# B&R Automation Studio project Ironer_Line
Automation Studio 4.7.2.98; technology packages: mapp 5.11.2, mappView 5.11.3

## Configuration Config1

CPU X20CP0484, AutomationRuntime B4.73, Build 4.1.2, Safety 0.0, Vc V4.44.0

### Task classes (Cpu.sw)
```
Cyclic#4 (cycle 100000 us, tolerance 100000 us):
  Failsafe <- Failsafe.prg
Cyclic#7 (cycle 1000000 us, tolerance 1000000 us):
  Data_log_p <- Data_log_prog.prg
Binaries: arsvcreg, TCData, udbdef, mvLoader, ashwd, sysconf, ashwac, asfw, arconfig, Role, Config, iomap, User, ArCoal, ArFlatPrv, OpcUaMap
Libraries: AsZip, FileIO, runtime, MpData, DataObj, sys_lib, brsystem, MpBase, astime, AsIODiag, asieccon, arssl
```

### Hardware
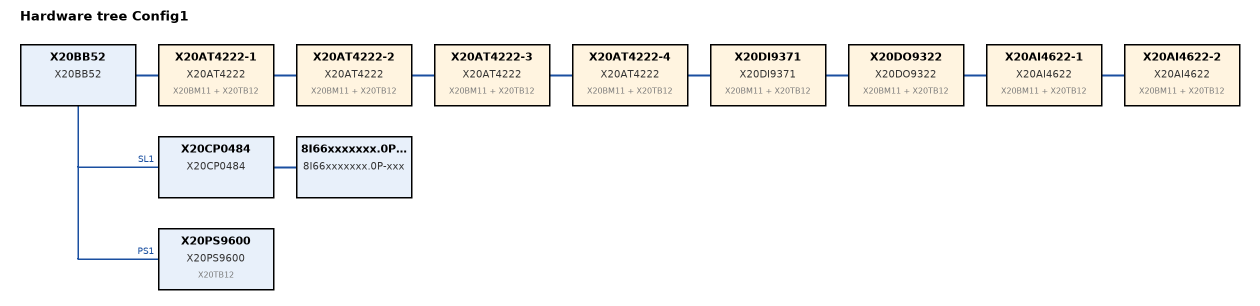
```
8I66xxxxxxx.0P-xxx : 8I66xxxxxxx.0P-xxx v2.3.0.0  [PLK1 -> X20CP0484.IF3 [Cable Type=PowerlinkCable, Length=10, Version=1.0.0.2]]
  FunctionModel = Standard
  Supervision = off
  UnitOfSetpoint = Rpm
  IOM_AIDP1 = ULN
  IOM_AIDP2 = RFR_D
  IOM_AIDP3 = UOP
  IOM_AIDP4 = LCR
  Sel_NameplateMask = MANU
  Cfg_NSP = 2853
  Cfg_UNS = 400
  Cfg_NCR = 25
  Cfg_COS = 80
  Cfg_NPR = 110
X20AI4622-1 : X20AI4622 v1.0.5.0  [SS1 -> X20TB12g.SS; SL -> X20BM11f.SL1]
  Supervision = off
  ChannelType01 = 4 to 20mA
X20AI4622-2 : X20AI4622 v1.0.5.0  [SS1 -> X20TB12h.SS; SL -> X20BM11g.SL1]
  Supervision = off
  ChannelType01 = 4 to 20mA
  ChannelType02 = 4 to 20mA
  ChannelType03 = 4 to 20mA
X20AT4222-1 : X20AT4222 v1.2.2.0  [SS1 -> X20TB12a.SS; SL -> X20BM11.SL1]
  FunctionModel = FunctionModel001
  Supervision = off
  SensorType02 = off
  SensorType03 = off
X20AT4222-2 : X20AT4222 v1.2.2.0  [SS1 -> X20TB12b.SS; SL -> X20BM11a.SL1]
  FunctionModel = FunctionModel001
  Supervision = off
  SensorType03 = off
  SensorType04 = off
X20AT4222-3 : X20AT4222 v1.2.2.0  [SS1 -> X20TB12c.SS; SL -> X20BM11b.SL1]
  FunctionModel = FunctionModel001
  Supervision = off
  SensorType03 = off
  SensorType04 = off
X20AT4222-4 : X20AT4222 v1.2.2.0  [SS1 -> X20TB12d.SS; SL -> X20BM11c.SL1]
  FunctionModel = FunctionModel001
  Supervision = off
  SensorType03 = off
  SensorType04 = off
X20BB52 : X20BB52 v1.1.0.0
X20BM11 : X20BM11 v1.0.0.1  [X2X1 -> X20BB52.IF6]
X20BM11a : X20BM11 v1.0.0.1  [X2X1 -> X20BM11.X2X2]
X20BM11b : X20BM11 v1.0.0.1  [X2X1 -> X20BM11a.X2X2]
X20BM11c : X20BM11 v1.0.0.1  [X2X1 -> X20BM11b.X2X2]
X20BM11d : X20BM11 v1.0.0.1  [X2X1 -> X20BM11c.X2X2]
X20BM11e : X20BM11 v1.0.0.1  [X2X1 -> X20BM11d.X2X2]
X20BM11f : X20BM11 v1.0.0.1  [X2X1 -> X20BM11e.X2X2]
X20BM11g : X20BM11 v1.0.0.1  [X2X1 -> X20BM11f.X2X2]
X20CP0484 : X20CP0484 v1.2.0.0  [SL -> X20BB52.SL1]
  Connector IF2:
    ActivateDevice = 1
    Mode = Manual
    InternetAddress = 10.0.0.2
    SubnetMask = 255.255.255.0
    InaNodeNumber = 0
  ConfigurationID = EIT5Projekt1_Config1
  UserPartitionSize = 100
  Simulation = 1
  TimerDeviceType = SWIOTIMER
  Cyclic1Duration = 10000
  Cyclic1Tolerance = 10000
  Cyclic2Duration = 20000
  Cyclic2Tolerance = 20000
  Cyclic3Duration = 50000
  Cyclic3Tolerance = 50000
  Cyclic4Duration = 100000
  Cyclic4Tolerance = 100000
  Cyclic5Duration = 200000
  Cyclic5Tolerance = 200000
  Cyclic6Duration = 500000
  Cyclic6Tolerance = 500000
  Cyclic7Duration = 1000000
  Cyclic7Tolerance = 1000000
  Cyclic8Duration = 10000
  Cyclic8Tolerance = 30000000
  FileDevice1
  FileDeviceName1 = PLC_user
  FileDevicePath1 = F:\
  FileDevice2
  FileDeviceName2 = PC_temp
  FileDevicePath2 = C:\temp\
  FtpUser1
  FtpUsername1 = admin
  FtpUserPassword1 = cwHDI+xQYJGOTM1OUrZCZFPwGlAu3H/MLCABeDPRdiI=  // password=admin
  FtpUserSalt1 = YD4DOUwF
  FTPAccessRight1 = 0
  FTPdevice1 = ALL
  ActivateOpcUa = 1
  OpcUaInformationModels_PV_Version = 1
X20DI9371 : X20DI9371 v1.0.2.0  [SS1 -> X20TB12e.SS; SL -> X20BM11d.SL1]
  Supervision = off
X20DO9322 : X20DO9322 v1.0.3.0  [SS1 -> X20TB12f.SS; SL -> X20BM11e.SL1]
  Supervision = off
X20PS9600 : X20PS9600 v1.0.1.0  [PS -> X20BB52.PS1; SS1 -> X20TB12.SS]
  Supervision = off
X20TB12 : X20TB12 v1.0.0.0
X20TB12a : X20TB12 v1.0.0.0
X20TB12b : X20TB12 v1.0.0.0
X20TB12c : X20TB12 v1.0.0.0
X20TB12d : X20TB12 v1.0.0.0
X20TB12e : X20TB12 v1.0.0.0
X20TB12f : X20TB12 v1.0.0.0
X20TB12g : X20TB12 v1.0.0.0
X20TB12h : X20TB12 v1.0.0.0
```

### IoMap.iom - X20CP0484/IoMap.iom
```iecst
VAR_CONFIG
	::T_tank AT %IW."X20AT4222-1".Temperature01;
	::inverter.CTRL_set AT %QW."8I66xxxxxxx.0P-xxx".CMDD_Output;
	::inverter.RPM_set AT %QW."8I66xxxxxxx.0P-xxx".LFRD_Output;
	::inverter.RPM_actual AT %IW."8I66xxxxxxx.0P-xxx".RFRD_Input;
	::inverter.freq AT %IW."8I66xxxxxxx.0P-xxx".RFR_Input;
	::inverter.voltage AT %IW."8I66xxxxxxx.0P-xxx".UOP_Input;
	::inverter.current AT %IW."8I66xxxxxxx.0P-xxx".LCR_Input;
	::inverter.DC AT %IW."8I66xxxxxxx.0P-xxx".ULN_Input;
	::inverter.error_code AT %IW."8I66xxxxxxx.0P-xxx".ERRD_Input;
	::inverter.CTRL_actual AT %IW."8I66xxxxxxx.0P-xxx".ETAD_Input;
	::inverter.RPM_after_ramp AT %IW."8I66xxxxxxx.0P-xxx".FROD_Input;
	::mulde_3.T_out AT %IW."X20AT4222-4".Temperature02;
	::mulde_3.T_in AT %IW."X20AT4222-4".Temperature01;
	::mulde_1.T_in AT %IW."X20AT4222-2".Temperature01;
	::mulde_2.T_out AT %IW."X20AT4222-3".Temperature02;
	::mulde_2.T_in AT %IW."X20AT4222-3".Temperature01;
	::mulde_1.T_out AT %IW."X20AT4222-2".Temperature02;
	::heater AT %QX."X20DO9322".DigitalOutput01;
	::T_ambient AT %IW."X20AT4222-1".Temperature04;
	::flow_cooling_water AT %IW."X20AI4622-1".AnalogInput01;
	::p_pumpe.before AT %IW."X20AI4622-2".AnalogInput01;
	::p_pumpe.after AT %IW."X20AI4622-2".AnalogInput02;
	::p_last AT %IW."X20AI4622-2".AnalogInput03;
END_VAR
```

### Config.mpdatarecorder - X20CP0484/mappServices/Config.mpdatarecorder
```
Element gDataRecorder (Type=mpdatarecorder)
  DataRecorder:
    MaxNumberOfFiles = 100
    MaxFileSize = 51200
```

## Logical view

Binary libraries used (declarations not repeated): operator, runtime, astime, AsIecCon, AsZip, FileIO, DataObj, sys_lib, brsystem, MpData 5.11.2, MpBase 5.11.0, AsIODiag

### Global.typ - Global data types
```iecst
TYPE
	inverter_type : 	STRUCT
		CTRL_set : UINT;
		CTRL_actual : UINT;
		RPM_set : INT;
		RPM_actual : INT;
		RPM_after_ramp : INT;
		error_code : UINT;
		freq : INT;
		voltage : UINT;
		current : UINT;
		DC : UINT;
	END_STRUCT;
	mulde_type : 	STRUCT
		olie : olie_type;
		toej : toej_type;
	END_STRUCT;
	p_pumpe_type : 	STRUCT
		after : INT;
		before : INT;
	END_STRUCT;
	olie_type : 	STRUCT
		T_out : INT;
		T_in : INT;
	END_STRUCT;
	toej_type : 	STRUCT
		T_out : INT;
		T_in : INT;
	END_STRUCT;
END_TYPE
```

### Global.var - Global variables
```iecst
VAR
	flow_cooling_water : INT;
	failState : UINT := 0;
	T_ambient : INT;
	mulde_3 : mulde_type;
	mulde_2 : mulde_type;
	mulde_1 : mulde_type;
	inverter : inverter_type;
	p_pumpe : p_pumpe_type;
	T_tank : INT;
	heater : BOOL;
	p_last : INT;
END_VAR
```


### Program Logical/Data_log_prog (IEC)

#### Main.st - Init, cyclic, exit code
```iecst
PROGRAM _INIT
	inverter;
	T_tank;
	T_ambient;
	heater;
	mulde_1;
	mulde_2;
	mulde_3;
	flow_cooling_water;
	p_pumpe;
	p_last;

	IF DiagCpuIsSimulated() THEN
		DataRecorder.DeviceName := ADR('PC_temp');
	ELSE
		DataRecorder.DeviceName := ADR('PLC_user');
	END_IF

	DataRecorder.MpLink := ADR(gDataRecorder);
	DataRecorder.RecordMode := mpDATA_RECORD_MODE_TIME;
	DataRecorder.SamplingTime := T#1s;

	DRP_T_ambient.MpLink := ADR(gDataRecorder);
	DRP_T_ambient.PVName := ADR('T_ambient'); //LOCAL variable:  Data_log_p:T_ambient

	DRP_heater.MpLink := ADR(gDataRecorder);
	DRP_heater.PVName := ADR('heater');

	DRP_T_tank.MpLink := ADR(gDataRecorder);
	DRP_T_tank.PVName := ADR('T_tank');

	DRP_inverter_RPM.MpLink := ADR(gDataRecorder);
	DRP_inverter_RPM.PVName := ADR('inverter.RPM_actual');

	DRP_m1_olie_Ti.MpLink := ADR(gDataRecorder);
	DRP_m1_olie_Ti.PVName := ADR('mulde_1.olie.T_in');

	DRP_m1_olie_To.MpLink := ADR(gDataRecorder);
	DRP_m1_olie_To.PVName := ADR('mulde_1.olie.T_out');

	DRP_m2_olie_Ti.MpLink := ADR(gDataRecorder);
	DRP_m2_olie_Ti.PVName := ADR('mulde_2.olie.T_in');

	DRP_m2_olie_To.MpLink := ADR(gDataRecorder);
	DRP_m2_olie_To.PVName := ADR('mulde_2.olie.T_out');

	DRP_m3_olie_Ti.MpLink := ADR(gDataRecorder);
	DRP_m3_olie_Ti.PVName := ADR('mulde_3.olie.T_in');

	DRP_m3_olie_To.MpLink := ADR(gDataRecorder);
	DRP_m3_olie_To.PVName := ADR('mulde_3.olie.T_out');

	DRP_p_pumpe_before.MpLink := ADR(gDataRecorder);
	DRP_p_pumpe_before.PVName := ADR('p_pumpe.before');

	DRP_p_pumpe_after.MpLink := ADR(gDataRecorder);
	DRP_p_pumpe_after.PVName := ADR('p_pumpe.after');

	DRP_p_last.MpLink := ADR(gDataRecorder);
	DRP_p_last.PVName := ADR('p_last');

	DRP_inverter_DC.MpLink := ADR(gDataRecorder);
	DRP_inverter_DC.PVName := ADR('inverter.DC');

	DRP_inverter_voltage.MpLink := ADR(gDataRecorder);
	DRP_inverter_voltage.PVName := ADR('inverter.voltage');

	DRP_inverter_current.MpLink := ADR(gDataRecorder);
	DRP_inverter_current.PVName := ADR('inverter.current');

	DRP_m1_toej_Ti.MpLink := ADR(gDataRecorder);
	DRP_m1_toej_Ti.PVName := ADR('mulde_1.toej.T_in');

	DRP_m1_toej_To.MpLink := ADR(gDataRecorder);
	DRP_m1_toej_To.PVName := ADR('mulde_1.toej.T_out');

	DRP_m2_toej_Ti.MpLink := ADR(gDataRecorder);
	DRP_m2_toej_Ti.PVName := ADR('mulde_2.toej.T_in');

	DRP_m2_toej_To.MpLink := ADR(gDataRecorder);
	DRP_m2_toej_To.PVName := ADR('mulde_2.toej.T_out');

	DRP_m3_toej_Ti.MpLink := ADR(gDataRecorder);
	DRP_m3_toej_Ti.PVName := ADR('mulde_3.toej.T_in');

	DRP_m3_toej_To.MpLink := ADR(gDataRecorder);
	DRP_m3_toej_To.PVName := ADR('mulde_3.toej.T_out');

	DRP_failState.MpLink := ADR(gDataRecorder);
	DRP_failState.PVName := ADR('failState');

	DRP_flow_cooling_water.MpLink := ADR(gDataRecorder);
	DRP_flow_cooling_water.PVName := ADR('flow_cooling_water');

	DRP_ctrl_ref.MpLink := ADR(gDataRecorder);
	DRP_ctrl_ref.PVName := ADR('Kontroller:ref');

	DRP_ctrl_D_u.MpLink := ADR(gDataRecorder);
	DRP_ctrl_D_u.PVName := ADR('Kontroller:D.u');

	DRP_PWM_duty.MpLink := ADR(gDataRecorder);
	DRP_PWM_duty.PVName := ADR('Kontroller:PWM.duty');

END_PROGRAM

PROGRAM _CYCLIC

	CASE state OF

		0:
			DataRecorder.Enable := TRUE;

			IF DataRecorder.Active AND NOT DataRecorder.CommandBusy THEN
				IF DataRecorder.StatusID = 0 THEN
					state := 10;
				ELSE
					state := 200;
				END_IF
			END_IF

		10:
			DRP_T_ambient.Enable := TRUE;

			IF DRP_T_ambient.Active THEN
				IF DRP_T_ambient.StatusID = 0 THEN
					DRP_T_ambient.Enable := TRUE;
					state := 20;
				ELSE
					state := 200;
				END_IF
			END_IF

			DRP_heater.Enable := TRUE;

			IF DRP_heater.Active THEN
				IF DRP_heater.StatusID = 0 THEN
					DRP_heater.Enable := TRUE;
					state := 20;
				ELSE
					state := 200;
				END_IF
			END_IF

			DRP_inverter_RPM.Enable := TRUE;

			IF DRP_inverter_RPM.Active THEN
				IF DRP_inverter_RPM.StatusID = 0 THEN
					DRP_inverter_RPM.Enable := TRUE;
					state := 20;
				ELSE
					state := 200;
				END_IF
			END_IF

			DRP_T_tank.Enable := TRUE;

			IF DRP_T_tank.Active THEN
				IF DRP_T_tank.StatusID = 0 THEN
					DRP_T_tank.Enable := TRUE;
					state := 20;
				ELSE
					state := 200;
				END_IF
			END_IF

			DRP_m1_olie_Ti.Enable := TRUE;

			IF DRP_m1_olie_Ti.Active THEN
				IF DRP_m1_olie_Ti.StatusID = 0 THEN
					DRP_m1_olie_Ti.Enable := TRUE;
					state := 20;
				ELSE
					state := 200;
				END_IF
			END_IF

			DRP_m1_olie_To.Enable := TRUE;

			IF DRP_m1_olie_To.Active THEN
				IF DRP_m1_olie_To.StatusID = 0 THEN
					DRP_m1_olie_To.Enable := TRUE;
					state := 20;
				ELSE
					state := 200;
				END_IF
			END_IF

			DRP_m2_olie_Ti.Enable := TRUE;

			IF DRP_m2_olie_Ti.Active THEN
				IF DRP_m2_olie_Ti.StatusID = 0 THEN
					DRP_m2_olie_Ti.Enable := TRUE;
					state := 20;
				ELSE
					state := 200;
				END_IF
			END_IF

			DRP_m2_olie_To.Enable := TRUE;

			IF DRP_m2_olie_To.Active THEN
				IF DRP_m2_olie_To.StatusID = 0 THEN
					DRP_m2_olie_To.Enable := TRUE;
					state := 20;
				ELSE
					state := 200;
				END_IF
			END_IF

			DRP_m3_olie_Ti.Enable := TRUE;

			IF DRP_m3_olie_Ti.Active THEN
				IF DRP_m3_olie_Ti.StatusID = 0 THEN
					DRP_m3_olie_Ti.Enable := TRUE;
					state := 20;
				ELSE
					state := 200;
				END_IF
			END_IF

			DRP_m3_olie_To.Enable := TRUE;

			IF DRP_m3_olie_To.Active THEN
				IF DRP_m3_olie_To.StatusID = 0 THEN
					DRP_m3_olie_To.Enable := TRUE;
					state := 20;
				ELSE
					state := 200;
				END_IF
			END_IF

			DRP_p_pumpe_before.Enable := TRUE;

			IF DRP_p_pumpe_before.Active THEN
				IF DRP_p_pumpe_before.StatusID = 0 THEN
					DRP_p_pumpe_before.Enable := TRUE;
					state := 20;
				ELSE
					state := 200;
				END_IF
			END_IF

			DRP_p_pumpe_after.Enable := TRUE;

			IF DRP_p_pumpe_after.Active THEN
				IF DRP_p_pumpe_after.StatusID = 0 THEN
					DRP_p_pumpe_after.Enable := TRUE;
					state := 20;
				ELSE
					state := 200;
				END_IF
			END_IF

			DRP_p_last.Enable := TRUE;

			IF DRP_p_last.Active THEN
				IF DRP_p_last.StatusID = 0 THEN
					DRP_p_last.Enable := TRUE;
					state := 20;
				ELSE
					state := 200;
				END_IF
			END_IF

			DRP_inverter_DC.Enable := TRUE;

			IF DRP_inverter_DC.Active THEN
				IF DRP_inverter_DC.StatusID = 0 THEN
					DRP_inverter_DC.Enable := TRUE;
					state := 20;
				ELSE
					state := 200;
				END_IF
			END_IF

			DRP_inverter_voltage.Enable := TRUE;

			IF DRP_inverter_voltage.Active THEN
				IF DRP_inverter_voltage.StatusID = 0 THEN
					DRP_inverter_voltage.Enable := TRUE;
					state := 20;
				ELSE
					state := 200;
				END_IF
			END_IF

			DRP_inverter_current.Enable := TRUE;

			IF DRP_inverter_current.Active THEN
				IF DRP_inverter_current.StatusID = 0 THEN
					DRP_inverter_current.Enable := TRUE;
					state := 20;
				ELSE
					state := 200;
				END_IF
			END_IF

			DRP_m1_toej_Ti.Enable := TRUE;

			IF DRP_m1_toej_Ti.Active THEN
				IF DRP_m1_toej_Ti.StatusID = 0 THEN
					DRP_m1_toej_Ti.Enable := TRUE;
					state := 20;
				ELSE
					state := 200;
				END_IF
			END_IF

			DRP_m1_toej_To.Enable := TRUE;

			IF DRP_m1_toej_To.Active THEN
				IF DRP_m1_toej_To.StatusID = 0 THEN
					DRP_m1_toej_To.Enable := TRUE;
					state := 20;
				ELSE
					state := 200;
				END_IF
			END_IF

			DRP_m2_toej_Ti.Enable := TRUE;

			IF DRP_m2_toej_Ti.Active THEN
				IF DRP_m2_toej_Ti.StatusID = 0 THEN
					DRP_m2_toej_Ti.Enable := TRUE;
					state := 20;
				ELSE
					state := 200;
				END_IF
			END_IF

			DRP_m2_toej_To.Enable := TRUE;

			IF DRP_m2_toej_To.Active THEN
				IF DRP_m2_toej_To.StatusID = 0 THEN
					DRP_m2_toej_To.Enable := TRUE;
					state := 20;
				ELSE
					state := 200;
				END_IF
			END_IF

			DRP_m3_toej_Ti.Enable := TRUE;

			IF DRP_m3_toej_Ti.Active THEN
				IF DRP_m3_toej_Ti.StatusID = 0 THEN
					DRP_m3_toej_Ti.Enable := TRUE;
					state := 20;
				ELSE
					state := 200;
				END_IF
			END_IF

			DRP_m3_toej_To.Enable := TRUE;

			IF DRP_m3_toej_To.Active THEN
				IF DRP_m3_toej_To.StatusID = 0 THEN
					DRP_m3_toej_To.Enable := TRUE;
					state := 20;
				ELSE
					state := 200;
				END_IF
			END_IF

			DRP_failState.Enable := TRUE;

			IF DRP_failState.Active THEN
				IF DRP_failState.StatusID = 0 THEN
					DRP_failState.Enable := TRUE;
					state := 20;
				ELSE
					state := 200;
				END_IF
			END_IF

			DRP_flow_cooling_water.Enable := TRUE;

			IF DRP_flow_cooling_water.Active THEN
				IF DRP_flow_cooling_water.StatusID = 0 THEN
					DRP_flow_cooling_water.Enable := TRUE;
					state := 20;
				ELSE
					state := 200;
				END_IF
			END_IF

			DRP_ctrl_ref.Enable := TRUE;

			IF DRP_ctrl_ref.Active THEN
				IF DRP_ctrl_ref.StatusID = 0 THEN
					DRP_ctrl_ref.Enable := TRUE;
					state := 20;
				ELSE
					state := 200;
				END_IF
			END_IF

			DRP_ctrl_D_u.Enable := TRUE;

			IF DRP_ctrl_D_u.Active THEN
				IF DRP_ctrl_D_u.StatusID = 0 THEN
					DRP_ctrl_D_u.Enable := TRUE;
					state := 20;
				ELSE
					state := 200;
				END_IF
			END_IF

			DRP_PWM_duty.Enable := TRUE;

			IF DRP_PWM_duty.Active THEN
				IF DRP_PWM_duty.StatusID = 0 THEN
					DRP_PWM_duty.Enable := TRUE;
					state := 20;
				ELSE
					state := 200;
				END_IF
			END_IF

			// add more regpar in between..
		20:

			DataRecorder.Record := TRUE;

			IF DataRecorder.Recording THEN
				state := 30;
			END_IF

		30:

		200:

	END_CASE

	DataRecorder();
	DRP_T_ambient();
	DRP_heater();
	DRP_inverter_RPM();
	DRP_T_tank();
	DRP_m1_olie_Ti();
	DRP_m1_olie_To();
	DRP_m2_olie_Ti();
	DRP_m2_olie_To();
	DRP_m3_olie_Ti();
	DRP_m3_olie_To();
	DRP_p_pumpe_before();
	DRP_p_pumpe_after();
	DRP_p_last();
	DRP_inverter_DC();
	DRP_inverter_voltage();
	DRP_inverter_current();
	DRP_m1_toej_Ti();
	DRP_m1_toej_To();
	DRP_m2_toej_Ti();
	DRP_m2_toej_To();
	DRP_m3_toej_Ti();
	DRP_m3_toej_To();
	DRP_failState();
	DRP_flow_cooling_water();
	DRP_ctrl_ref();
	DRP_ctrl_D_u();
	DRP_PWM_duty();

END_PROGRAM

PROGRAM _EXIT

	DataRecorder(Enable := FALSE);
	DRP_T_ambient(Enable := FALSE);
	DRP_heater(Enable := FALSE);
	DRP_inverter_RPM(Enable := FALSE);
	DRP_T_tank(Enable := FALSE);
	DRP_m1_olie_Ti(Enable := FALSE);
	DRP_m1_olie_To(Enable := FALSE);
	DRP_m2_olie_Ti(Enable := FALSE);
	DRP_m2_olie_To(Enable := FALSE);
	DRP_m3_olie_Ti(Enable := FALSE);
	DRP_m3_olie_To(Enable := FALSE);
	DRP_p_pumpe_before(Enable := FALSE);
	DRP_p_pumpe_after(Enable := FALSE);
	DRP_p_last(Enable := FALSE);
	DRP_inverter_DC(Enable := FALSE);
	DRP_inverter_voltage(Enable := FALSE);
	DRP_inverter_current(Enable := FALSE);
	DRP_m1_toej_Ti(Enable := FALSE);
	DRP_m1_toej_To(Enable := FALSE);
	DRP_m2_toej_Ti(Enable := FALSE);
	DRP_m2_toej_To(Enable := FALSE);
	DRP_m3_toej_Ti(Enable := FALSE);
	DRP_m3_toej_To(Enable := FALSE);
	DRP_failState(Enable := FALSE);
	DRP_flow_cooling_water(Enable := FALSE);
	DRP_ctrl_ref(Enable := FALSE);
	DRP_ctrl_D_u(Enable := FALSE);
	DRP_PWM_duty(Enable := FALSE);

END_PROGRAM
```

#### Types.typ - Local data types
```iecst
TYPE
	STATE_ENUM :
		(
		STATE_RECORDING := 0
		);
END_TYPE
```

#### Variables.var - Local variables
```iecst
VAR
	DRP_inverter_voltage : MpDataRegPar;
	DRP_inverter_DC : MpDataRegPar;
	DRP_inverter_current : MpDataRegPar;
	DRP_inverter_RPM : MpDataRegPar;
	DataRecorder : MpDataRecorder;
	DRP_m3_toej_To : MpDataRegPar;
	DRP_m3_toej_Ti : MpDataRegPar;
	DRP_m2_toej_To : MpDataRegPar;
	DRP_m2_toej_Ti : MpDataRegPar;
	DRP_m1_toej_To : MpDataRegPar;
	DRP_m1_toej_Ti : MpDataRegPar;
	DRP_m3_olie_To : MpDataRegPar;
	DRP_m3_olie_Ti : MpDataRegPar;
	DRP_m2_olie_To : MpDataRegPar;
	DRP_m2_olie_Ti : MpDataRegPar;
	DRP_m1_olie_To : MpDataRegPar;
	DRP_m1_olie_Ti : MpDataRegPar;
	DRP_T_tank : MpDataRegPar;
	DRP_flow_cooling_water : MpDataRegPar;
	DRP_failState : MpDataRegPar;
	DRP_heater : MpDataRegPar;
	DRP_T_ambient : MpDataRegPar;
	state : USINT;
	DRP_p_pumpe_before : MpDataRegPar;
	DRP_p_pumpe_after : MpDataRegPar;
	DRP_PWM_duty : MpDataRegPar;
	DRP_ctrl_D_u : MpDataRegPar;
	DRP_ctrl_ref : MpDataRegPar;
	DRP_p_last : MpDataRegPar;
END_VAR
```

#### Cyclic.ld
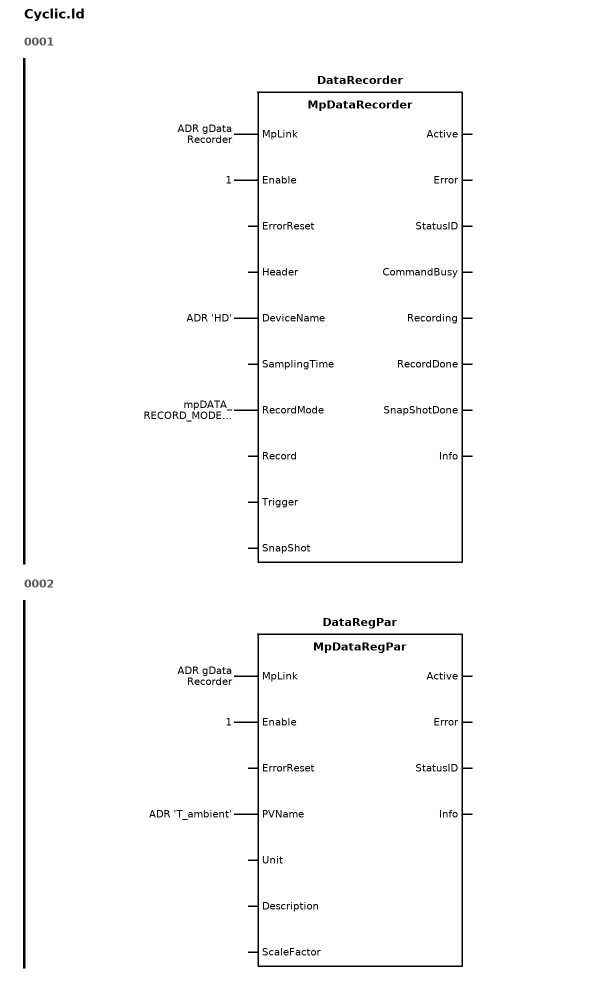
Ladder, written as Structured Text:
```iecst
PROGRAM _CYCLIC
(* Network 1 *)
DataRecorder(MpLink := ADR(gDataRecorder), Enable := 1, DeviceName := ADR('HD'), RecordMode := mpDATA_RECORD_MODE_VALUE);

(* Network 2 *)
DataRegPar(MpLink := ADR(gDataRecorder), Enable := 1, PVName := ADR('T_ambient'));
END_PROGRAM
```

- Visualisation Logical/mappView (not shown)

### Program Logical/Failsafe (ANSIC)

#### Types.typ - Local data types
```iecst
TYPE
	oc_type : 	STRUCT  (*over current protection type*)
		crb : ARRAY[0..299]OF UINT := [0]; (*Ring buffer for current. Acts as sample window*)
		avg : UINT := 0; (*average current inside sample window*)
		sum : UINT := 0; (*used for calculating the sum of the ring buffer*)
		N : UINT := 300; (*Length of ring buffer*)
		rp : UINT := 0; (*pointer for ringbuffer*)
		max : UINT := 25; (*maximum average current in dA*)
	END_STRUCT;
	tl_type : 	STRUCT  (*temperature limit type*)
		max : INT := 650; (*maximum temperature allowed in d°C*)
	END_STRUCT;
	hna_type : 	STRUCT  (*heater may not be on alone type*)
		cntr : UINT := 0; (*To count time*)
		minRPM : UINT := 500; (*minimum allowed RPM of pump*)
		timeout : UINT := 2400; (*in seconds times cycline period*)
	END_STRUCT;
	op_type : 	STRUCT  (*over pressure protection type*)
		max : REAL := 1.5; (*maximum pressure allowed in Bar*)
		P : REAL := 0.0; (*actual pressure (for calculations)*)
	END_STRUCT;
END_TYPE
```

#### Main.c - Init, cyclic, exit code
```c
#include <bur/plctypes.h>

#ifdef _DEFAULT_INCLUDES
	#include <AsDefault.h>
#endif

void _INIT ProgramInit(void)
{
	heater;
	inverter;
	mulde_1;
	mulde_2;
	mulde_3;
	p_last;
	p_pumpe;
	T_ambient;
	T_tank;

	failState;
	ocp;
	hna;
	tl;
}

void _CYCLIC ProgramCyclic(void)
{

	// To safely run code, only execute code if failState is 0!!! //

	failState | checkOverCurrent();
	failState | checkHeater();
	failState | checkTemperature();
	// add more check here //

	if (failstate != 0) {
		// something is wrong i can feel it
		// better shut down
		saveShutdown();
	}
	else {
		// everything is OK
	}

}

int checkOverCurrent(void) {

	// over current protection
	ocp.sum -= ocp.crb[ocp.rp]; //remove oldes current from sum
	ocp.sum += inverter.current; // add new current to sum
	ocp.crb[ocp.rp] = inverter.current; // add new current to ring buffer

	ocp.rp++; // increment ring buffer pointer
	if (ocp.rp >= ocp.N) {
		ocp.rp = 0; // overflow ring buffer pointer
	}

	ocp.avg = ocp.sum/(ocp.N); // calculate avg og ring buffer
	if (ocp.avg > ocp.max) {
		return 0x0001; // the average current was too high inside of sample window
	}
	else {
		return 0x0000; // no fail (overcurrent)
	}
}

int checkHeater(void) {

	// checks if heater is on for extended periods of time without flow in the system

	if (heater == 1 && inverter.RPM_actual < hna.minRPM){
		hna.cntr++;
	}
	else {
		hna.cntr = 0;
	}

	if (hna.cntr > hna.timeout) {
		return 0x0002;
	}
	else {
		return 0x0000;
	}
}

int checkTemperature(void) {

	// checks if any temperature is higher then allowed

	if(T_tank > tl.max) {
		return 0x0004;
	}
	else {
		return 0x0000;
	}
}

void saveShutdown(void) {

	inverter.RPM_set = 0;
	heater = 0;

}

void _EXIT ProgramExit(void)
{

}
```

#### Variables.var - Local variables
```iecst
VAR
	ocp : oc_type; (*over current protection struct*)
	hna : hna_type; (*heater not alone struct*)
	tl : tl_type; (*temperature limit struct*)
	opp : op_type; (*over pressure protection struct*)
END_VAR
```

### Program Logical/Kontroller (ANSIC)

#### Types.typ
```iecst
TYPE
	aaFilter_type : 	STRUCT  (*Anti aliasing filter*)
		timescale : UINT := 6;
		cntr : UINT := 0;
		a : ARRAY[0..2]OF LREAL; (*numerators*)
		b : ARRAY[0..2]OF LREAL; (*denumenators*)
		w : ARRAY[0..2]OF LREAL := [0];
	END_STRUCT;
	onOff_type : 	STRUCT
		dT : ARRAY[0..1]OF UINT; (*hysterese interval*)
	END_STRUCT;
	controller_type : 	STRUCT  (*Coefficients and registers for the kontroller*)
		e : LREAL; (*error signal*)
		b : ARRAY[0..2]OF LREAL; (*numerators of the discrete time transfer function*)
		a : ARRAY[0..2]OF LREAL; (*denuminator of the discrete time transfer function*)
		w : ARRAY[0..2]OF LREAL := [0]; (*intermediate signal for direct form II calculations*)
		offset : UINT := 918; (*Operating point offset*)
		u : LREAL; (*controller output*)
	END_STRUCT;
	PWM_type : 	STRUCT
		cntr : UINT := 0;
		timescale : UINT := 1000; (*used for scaling the sample time*)
		Pmax : REAL := 5200; (*maximum possible power*)
		duty : INT := 0; (*duty cycle*)
		out : BOOL := 0; (*PWM output to heater*)
	END_STRUCT;
END_TYPE
```

#### Variables.var
```iecst
VAR
	D : controller_type; (*coefficients and registers for the controller*)
	PWM : PWM_type; (*PWM parameters*)
	onOff : onOff_type; (*parameters for the onOff controller*)
	en : UINT := 0; (*do function variable*)
	ref : UINT := 100; (*referance signal in d°C*)
	T : UINT := 0; (*actual temperature in d°C*)
	en_last : UINT := 0; (*do function variable from last cycle*)
	aaF : aaFilter_type; (*anti aliasing filter*)
END_VAR
```

#### Main.c
```c
#include <bur/plctypes.h>

#ifdef _DEFAULT_INCLUDES
#include <AsDefault.h>
#endif

void contAlg(REAL e) {

	// implementation of the difference equations
	D.w[0] = D.a[0]*e - D.a[1]*D.w[1] - D.a[2]*D.w[2];
	D.u = D.b[0]*D.w[0] + D.b[1]*D.w[1] + D.b[2]*D.w[2];
	D.u += D.offset;

	// update of registers (delayed signals)
	D.w[2] = D.w[1];
	D.w[1] = D.w[0];

}

void PWM_fun(void) {

	en = 0;
	PWM.cntr++;

	if (PWM.cntr >= PWM.timescale + 1) { // +1 to not skip the last cycle
		en = 1; // do controller
		T = mulde_1.olie.T_in; // read measured temperature
		PWM.cntr = 0;
	}

	PWM.out = (PWM.cntr < PWM.duty); // set PWM out to true if cntr is smaller than dutycycle

}

void onOff_fun(void) {

	if (en==1) { // selects which controller to use
		if((T < (ref-onOff.dT[1])) || (T > (ref + onOff.dT[1]))) {
			en += 1; // use on-off controller
			en_last = en;
		}
		else if((T < (ref + onOff.dT[0])) && (T > (ref-onOff.dT[0]))) {
			en += 2; // use small-signal controller
			en_last = en;
		}
		else {
			en = en_last;
		}

	}

}

void D_fun(void) {

	if(en==2) { // do on-off controller
		D.e = 0;
		contAlg(D.e); // call controller to let it settle

		if(T < ref) {
			PWM.duty = PWM.timescale; // duty = timescale gives maximum output power
		}
		else {
			PWM.duty = 0;
		}
	}
	else if(en==3) { // do small-signal controller
		D.e = ref-T;
		contAlg((REAL)D.e); // calculate the control signal u[n]

		PWM.duty = ((INT)D.u*PWM.timescale)/PWM.Pmax; // times with timescale first to avoid floor division problmes :(
	}

}

void _INIT ProgramInit(void) {

	D;
	PWM;
	onOff;
	en;
	en_last;
	ref;
	T;

	// controller koefficients
	// denum
	D.a[0] = 1.00000;
	D.a[1] = -1.8568;
	D.a[2] = 0.8576;
	// num, divide by 10 because measured temp is in d°C
	D.b[0] = 140.74086 / 10;
	D.b[1] = 3.40703 / 10;
	D.b[2] = -137.33383 / 10;

	// hysterese interval
	onOff.dT[0] = 20;
	onOff.dT[1] = 40;

}

void _CYCLIC ProgramCyclic(void) {

	PWM_fun();
	onOff_fun();
	D_fun();

}

void _EXIT ProgramExit(void) {

}
```

### Program Logical/Omregner (ANSIC)

#### Variables.var
```iecst
VAR
	p_last_bar : REAL;
	p_after_pump_bar : REAL;
	p_before_pump_bar : REAL;
	flow_cooling_water_mls : REAL;
END_VAR
```

#### Main.c
```c
#include <bur/plctypes.h>

#ifdef _DEFAULT_INCLUDES
	#include <AsDefault.h>
#endif

void _INIT ProgramInit(void)
{

}

void _CYCLIC ProgramCyclic(void)
{

	p_before_pump_bar = (p_pumpe.before/32767.0)*10;
	p_after_pump_bar = (p_pumpe.after/32767.0)*10;
	p_last_bar = (p_last/32767.0)*10;
	flow_cooling_water_mls = (flow_cooling_water/32767.0)*500;

}

void _EXIT ProgramExit(void)
{

}
```

### Program Logical/Program (IEC)

#### Main.st - Init, cyclic, exit code
```iecst
PROGRAM _INIT
	inverter;
	T_tank;
	heater;
	mulde_1;
	mulde_2;
	mulde_3;

END_PROGRAM

PROGRAM _CYCLIC

END_PROGRAM

PROGRAM _EXIT

END_PROGRAM
```

#### Variables.var - Local variables
```iecst
VAR
	T : INT;
END_VAR
```

Listed in the project but not available here: Logical/Program/Types.typ
